// TIA Portal V15.1 export
// export: Created 2024-05-17T05:38:39.6404684Z, ExportSetting WithDefaults, DisplayName Totally Integrated Automation Portal, DisplayVersion V15.1 Update 5, DisplayName TIA Portal Openness, DisplayVersion V15.1 Update 5, DisplayName SINAMICS Startdrive Advanced, DisplayVersion V15.1, DisplayName G130, G150, S120, S150, SINAMICS MV, S210, DisplayVersion V15.1, DisplayName G110M, G120, G120C, G120D, G120P, DisplayVersion V15.1, DisplayName STEP 7 Professional, DisplayVersion V15.1 Update 5, DisplayName STEP 7 Safety, DisplayVersion V15.1, DisplayName WinCC Professional, DisplayVersion V15.1 Update 5, DisplayName SIMATIC Visualization Architect, DisplayVersion V15.1
FUNCTION_BLOCK "LGBCalcInc"   // FB6655, SCL
TITLE = 'L_LineFeedGC' / PTCConvCalcInc
{ S7_Optimized_Access := 'TRUE' }
AUTHOR : Imtech
FAMILY : Conv
VERSION : 0.1
// //In tracking-stations you normally use a fast counting-card to count the
// //conveyor-pulses. The length-increment - the way the conveyor moved since
// //the last block-cycle - is calculated by means of a coveyor-scaling-factor.
// //You can use this FB to calc the length increment.
// //
// //HANDLED SITUATIONS:
// //- pulse-peak detection - unnormal high pulse-peaks will be ignored and cause a
// //  reset
// //- counting forward, counting backward
// //- overflow handling forward/backward at 2147483647/-2147483647
// //- no division-error (division-remainder is considered in next cycle)
// //
// //INSTRUCTIONS:
// //- init/reset with a rising edge on "i_mRun" or "i_mReset". The current conveyor
// //  pulse count will be saved (internal) to avoid a pulse-peak
// //- set the value of the conveyor-counting-var as input-parameter of this FB
// //- set the max tolerable pulse-peak between two cycles as input-parameter
// //  for error-detection (approx. 4-10 times higher than the normal amount of
// //  pulses per cycle).
// //
// //SPEED CALCULATION:
// //The speed will be updated with a time-interval, which can be defined with the 
// //parameter "i_tSpeedCalcIntvl". Note: If you have a fast counting card the 
// //time-parameter may be low (e.g. 1-2s) so you get a fast update of the calculated
// //speed. If you have a slow counting-card (e.g. with impulse-division-card) you
// //should use a higher time-value. Of course the update of the time-value will
// //be more slow.
// //
// //CONVEYOR RUNNING:
// //The output-parameter "conveyor-running" is true, when the calculated conveyor-
// //increments are unequal to zero. This signal will be debounced with the time-
// //parameter "i_tConvRunDeb".
// stored: AutoNumber false, IsIECCheckEnabled false, IsRetainMemResEnabled false, MemoryReserve 100, SetENOAutomatically False, UDAEnableTagReadback false
   VAR_INPUT
      I_mRun { ExternalAccessible := 'False'; ExternalVisible := 'False'; ExternalWritable := 'False'} : Bool;   // enable FB and calc increments
      i_mReset { ExternalAccessible := 'False'; ExternalVisible := 'False'; ExternalWritable := 'False'} : Bool;   // reset/init FB
      i_tConvRunDeb { ExternalAccessible := 'False'; ExternalVisible := 'False'; ExternalWritable := 'False'} : Time := T#1s;   // debounce-time for signal "conveyor is running"
      i_tSpeedCalcIntvl { ExternalAccessible := 'False'; ExternalVisible := 'False'; ExternalWritable := 'False'} : Time := T#2s;   // update-interval for speed-calculation
      i_dMaxPulsePeak { ExternalAccessible := 'False'; ExternalVisible := 'False'; ExternalWritable := 'False'} : DInt;   // max. tolerable pulse-peak between two cycles (error detection)
      i_dPulseCount { ExternalAccessible := 'False'; ExternalVisible := 'False'; ExternalWritable := 'False'} : DInt;   // current value of pulse-counting-variable
      i_dScalingFactor { ExternalAccessible := 'False'; ExternalVisible := 'False'; ExternalWritable := 'False'} : DInt;   // scaling-factor [pulses/cm], > 0
   END_VAR
   VAR_OUTPUT
      o_iConvInc { ExternalAccessible := 'False'; ExternalVisible := 'False'; ExternalWritable := 'False'} : Int;   // length-increment since last cycle [cm]
      o_iSpeed { ExternalAccessible := 'False'; ExternalVisible := 'False'; ExternalWritable := 'False'} : Int;   // current conveyor-speed [cm/min]
      o_mConvRun { ExternalAccessible := 'False'; ExternalVisible := 'False'; ExternalWritable := 'False'} : Bool;   // conveyor is running (debounced signal)
      o_mErrPulsePeak { ExternalAccessible := 'False'; ExternalVisible := 'False'; ExternalWritable := 'False'} : Bool;   // error: an intolerable pulse-peak was detected
      o_mErrScalingFactor { ExternalAccessible := 'False'; ExternalVisible := 'False'; ExternalWritable := 'False'} : Bool;   // error: invalid scaling-factor
   END_VAR
   VAR
      dPulseCountOld { ExternalAccessible := 'False'; ExternalVisible := 'False'; ExternalWritable := 'False'} : DInt;   // last pulse-count
      dDivRemainder { ExternalAccessible := 'False'; ExternalVisible := 'False'; ExternalWritable := 'False'} : DInt;   // division-remainder for next cylce
      dPulsesSum { ExternalAccessible := 'False'; ExternalVisible := 'False'; ExternalWritable := 'False'} : DInt;   // pulses since last update-interval for speed-calculation
      mRunOld { ExternalAccessible := 'False'; ExternalVisible := 'False'; ExternalWritable := 'False'} : Bool;   // edge-detection
      fbTofConvRun { ExternalAccessible := 'False'; ExternalVisible := 'False'; ExternalWritable := 'False'} : TOF_TIME;   // delay-off for debouncing of signal "conveyor is running"
      fbTonConvSpeed { ExternalAccessible := 'False'; ExternalVisible := 'False'; ExternalWritable := 'False'} : TON_TIME;   // delaytimer to measure conveyor-speed
      rSpeed { ExternalAccessible := 'False'; ExternalVisible := 'False'; ExternalWritable := 'False'} : Real;   // speed as real-value
      rSpeedOld { ExternalAccessible := 'False'; ExternalVisible := 'False'; ExternalWritable := 'False'} : Real;   // old speed for speed averaging
   END_VAR
   VAR_TEMP
      dDeltaPulses : DInt;   // pulse-difference to last cycle [pulses]
      dSpeedCalcInterval : DInt;   // update-interval for speed-calculation [ms]
      dConvSum_fine : DInt;   // conveyor-distance [cm/60000] since last speed-calculation
      tSpeedCalcIntvl : Time;   // update-interval for speed-calculation
   END_VAR
   VAR CONSTANT
      cMinSpeedCalcInv1 : Time := T#1s;   // Minimum update-interval for speed calculation
      cMaxSpeedCalcInv1 : Time := T#20s;   // Maximum update-interval for speed calculation
   END_VAR
BEGIN
   //reset when reset or rising-edge of i_mRun
   IF #i_mReset OR (#I_mRun AND NOT #mRunOld) THEN

       //output-parameters
       #o_iConvInc := 0;
       #o_iSpeed := 0;
       #o_mErrPulsePeak := FALSE;
       #o_mErrScalingFactor := FALSE;

       //static vars
       #dPulseCountOld := #i_dPulseCount;
       #dDivRemainder := 0;
       #dPulsesSum := 0;
       RESET_TIMER("TIMER" := #fbTofConvRun);
       RESET_TIMER("TIMER" := #fbTonConvSpeed);

       #rSpeed := 0.0;
       #rSpeedOld := 0.0;

   END_IF;
   #mRunOld := #I_mRun; //edge-detection


   //exit when not i_mRun
   IF NOT #I_mRun THEN
       #o_iConvInc := 0;      //clear output
       #o_iSpeed := 0;
       RETURN;
   END_IF;


   //calc pulse-difference
   (*
   - consider overflow-situations (overflow forward, overflow backward)
   - check for pulse-peak
   *)
   #dDeltaPulses := #i_dPulseCount - #dPulseCountOld;

   IF (#dDeltaPulses <= #i_dMaxPulsePeak)      //normal forward
       AND (#dDeltaPulses >= - #i_dMaxPulsePeak) THEN //normal backward
       ;

   ELSIF (#dDeltaPulses <= (-2147483647 + #i_dMaxPulsePeak)) THEN    //overflow forward

       #dDeltaPulses := #dDeltaPulses + 2147483647;

   ELSIF (#dDeltaPulses >= (2147483647 - #i_dMaxPulsePeak)) THEN     //overflow backward

       #dDeltaPulses := #dDeltaPulses - 2147483647;

   ELSE

       #o_mErrPulsePeak := TRUE;            //set error
       #o_iConvInc := 0;               //clear output
       #o_iSpeed := 0;
       #dPulseCountOld := #i_dPulseCount;   //init conveyor pulse-count
       #dPulsesSum := 0;
       RETURN;

   END_IF;

   //check scaling-factor
   IF #i_dScalingFactor <= 0 THEN

       #o_mErrScalingFactor := TRUE;    //set error
       #o_iConvInc := 0;       //clear output
       #o_iSpeed := 0;
       RETURN;

   ELSE
       #o_mErrScalingFactor := FALSE;   //reset error
   END_IF;


   //calc conveyor-length-increment
   #o_iConvInc := DINT_TO_INT(((#dDeltaPulses) + #dDivRemainder) / #i_dScalingFactor);

   //save division-remainder for next cycle
   #dDivRemainder := ((#dDeltaPulses) + #dDivRemainder) MOD #i_dScalingFactor;



   //calc conveyor-speed -------------------------------------------------------------------------------------------------

   //sum conveyor-pulses
   #dPulsesSum := #dPulsesSum + #dDeltaPulses;

   //copy update-interval to local-temp for better performance           
   #tSpeedCalcIntvl := #i_tSpeedCalcIntvl;

   //correct update-interval for speed-calculation if necessary
   IF #tSpeedCalcIntvl > #cMaxSpeedCalcInv1 THEN
       #tSpeedCalcIntvl := #cMaxSpeedCalcInv1;
   ELSIF #tSpeedCalcIntvl < #cMinSpeedCalcInv1 THEN
       #tSpeedCalcIntvl := #cMinSpeedCalcInv1;
   END_IF;

   //SPEED CALCULATION: update timer
   #fbTonConvSpeed(IN := TRUE,
                   PT := #cMaxSpeedCalcInv1);

   //SPEED CALCULATION: check if update-time is reached               
   IF #fbTonConvSpeed.ET >= #tSpeedCalcIntvl THEN

       //calculate speed on used time-base
       #dSpeedCalcInterval := TIME_TO_DINT(#fbTonConvSpeed.ET);  //convert time to DINT (e.a. T#2530ms -> 2530). Use x.ET directly for better accurracy
       #rSpeed := (DINT_TO_REAL(#dPulsesSum) * 60000.0) /        //calc speed: dSpeedCalcInterval has unit [ms]. Multiplied with 60000 results unit [min]
       DINT_TO_REAL((#i_dScalingFactor * #dSpeedCalcInterval));

       #o_iSpeed := REAL_TO_INT((#rSpeed + #rSpeedOld) / 2.0);   //calc averaged speed (speed of this cycle + speed of last cycle) / 2
       #rSpeedOld := #rSpeed;                                    //save speed of this cycle for next cycle
       #dPulsesSum := 0;                                       //init for new speed calculation

       //reset timer
       #fbTonConvSpeed(IN := FALSE,
                       PT := T#0s);

   END_IF;

   #fbTonConvSpeed(IN := TRUE,
                   PT := #cMaxSpeedCalcInv1);


   //generate signal "conveyor is running"
   #fbTofConvRun(IN := (#o_iConvInc <> 0),
                 PT := #i_tConvRunDeb);

   #o_mConvRun := #fbTofConvRun.Q;


   #dPulseCountOld := #i_dPulseCount;    //save pulse-count for next cycle
END_FUNCTION_BLOCK
